// Mitsubishi GX Works2 project: 4way-intersection   PLC: Q03UDV

PROGRAM MAIN
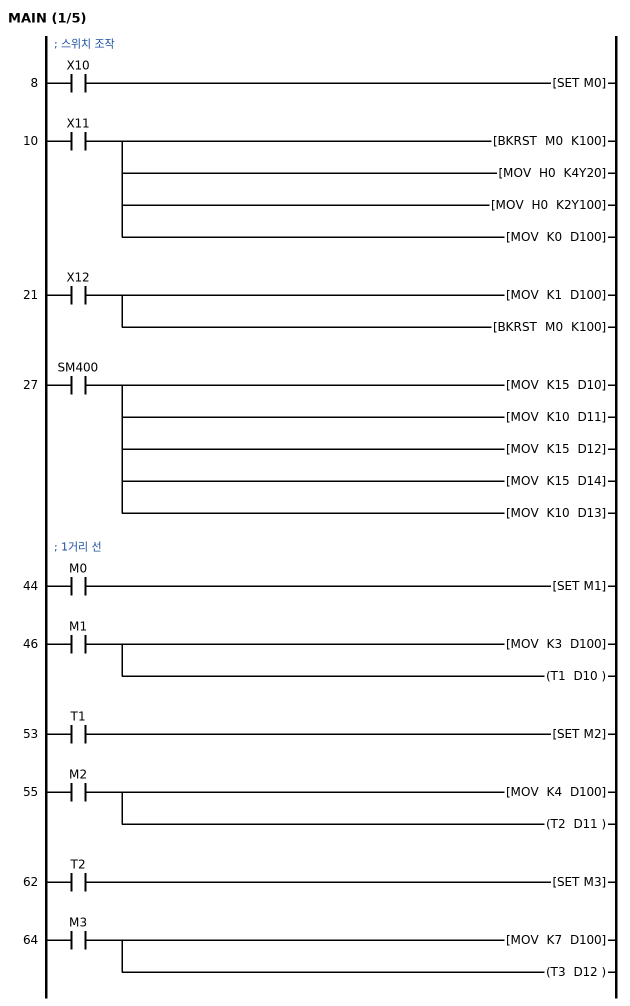
; 스위치 조작
8     LD      X10
      SET     M0
10    LD      X11
      BKRST   M0 K100
      MOV     H0 K4Y20
      MOV     H0 K2Y100
      MOV     K0 D100
21    LD      X12
      MOV     K1 D100
      BKRST   M0 K100
27    LD      SM400
      MOV     K15 D10
      MOV     K10 D11
      MOV     K15 D12
      MOV     K15 D14
      MOV     K10 D13
; 1거리 선
44    LD      M0
      SET     M1
46    LD      M1
      MOV     K3 D100
      OUT     T1 D10
53    LD      T1
      SET     M2
55    LD      M2
      MOV     K4 D100
      OUT     T2 D11
62    LD      T2
      SET     M3
64    LD      M3
      MOV     K7 D100
      OUT     T3 D12
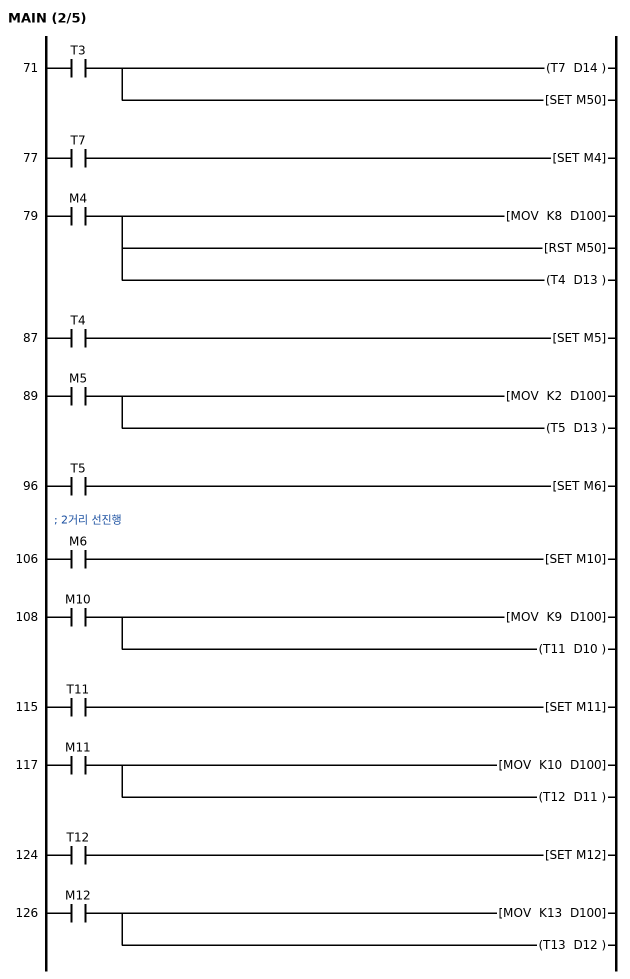
71    LD      T3
      OUT     T7 D14
      SET     M50
77    LD      T7
      SET     M4
79    LD      M4
      MOV     K8 D100
      RST     M50
      OUT     T4 D13
87    LD      T4
      SET     M5
89    LD      M5
      MOV     K2 D100
      OUT     T5 D13
96    LD      T5
      SET     M6
; 2거리 선진행
106   LD      M6
      SET     M10
108   LD      M10
      MOV     K9 D100
      OUT     T11 D10
115   LD      T11
      SET     M11
117   LD      M11
      MOV     K10 D100
      OUT     T12 D11
124   LD      T12
      SET     M12
126   LD      M12
      MOV     K13 D100
      OUT     T13 D12
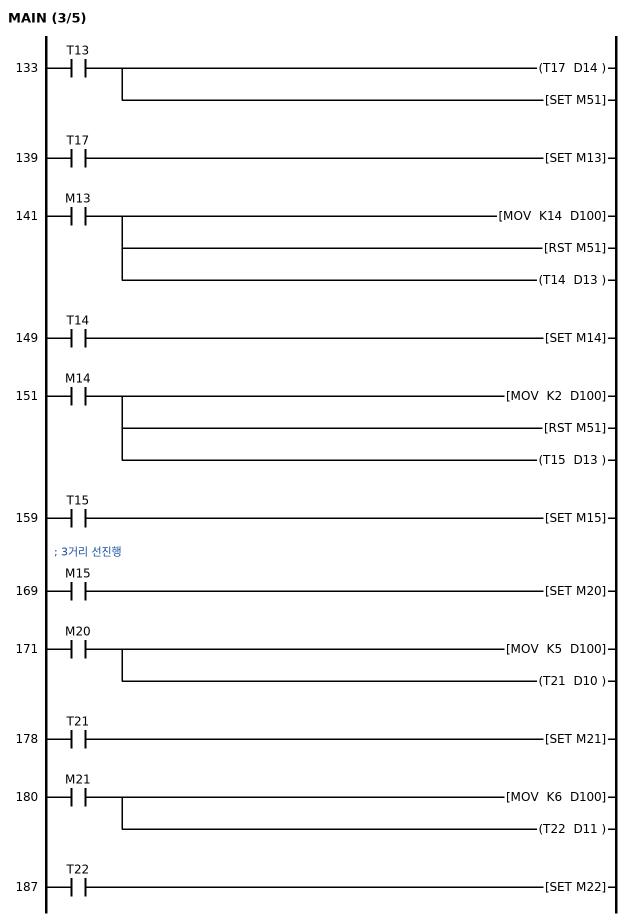
133   LD      T13
      OUT     T17 D14
      SET     M51
139   LD      T17
      SET     M13
141   LD      M13
      MOV     K14 D100
      RST     M51
      OUT     T14 D13
149   LD      T14
      SET     M14
151   LD      M14
      MOV     K2 D100
      RST     M51
      OUT     T15 D13
159   LD      T15
      SET     M15
; 3거리 선진행
169   LD      M15
      SET     M20
171   LD      M20
      MOV     K5 D100
      OUT     T21 D10
178   LD      T21
      SET     M21
180   LD      M21
      MOV     K6 D100
      OUT     T22 D11
187   LD      T22
      SET     M22
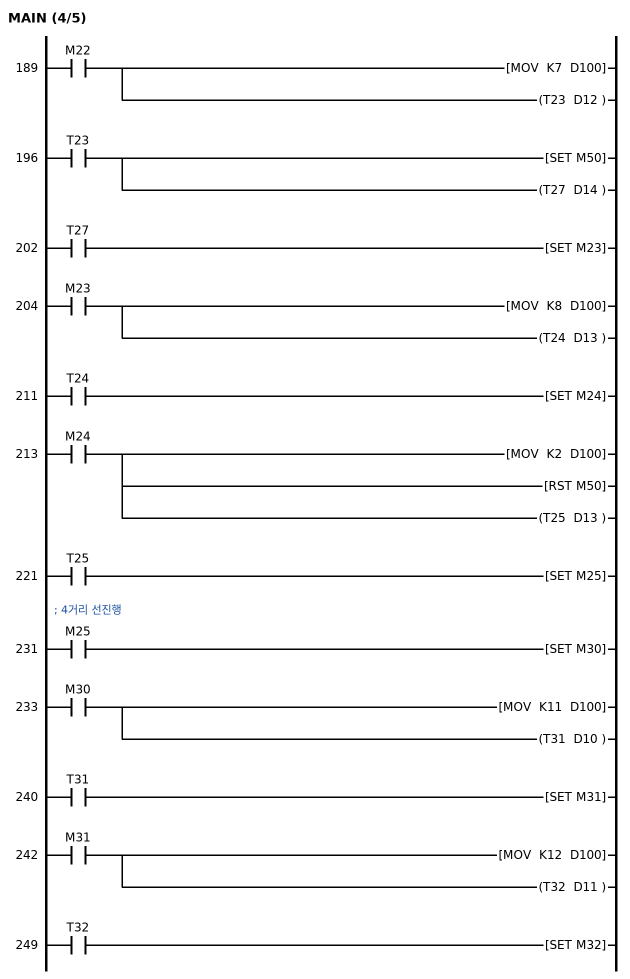
189   LD      M22
      MOV     K7 D100
      OUT     T23 D12
196   LD      T23
      SET     M50
      OUT     T27 D14
202   LD      T27
      SET     M23
204   LD      M23
      MOV     K8 D100
      OUT     T24 D13
211   LD      T24
      SET     M24
213   LD      M24
      MOV     K2 D100
      RST     M50
      OUT     T25 D13
221   LD      T25
      SET     M25
; 4거리 선진행
231   LD      M25
      SET     M30
233   LD      M30
      MOV     K11 D100
      OUT     T31 D10
240   LD      T31
      SET     M31
242   LD      M31
      MOV     K12 D100
      OUT     T32 D11
249   LD      T32
      SET     M32
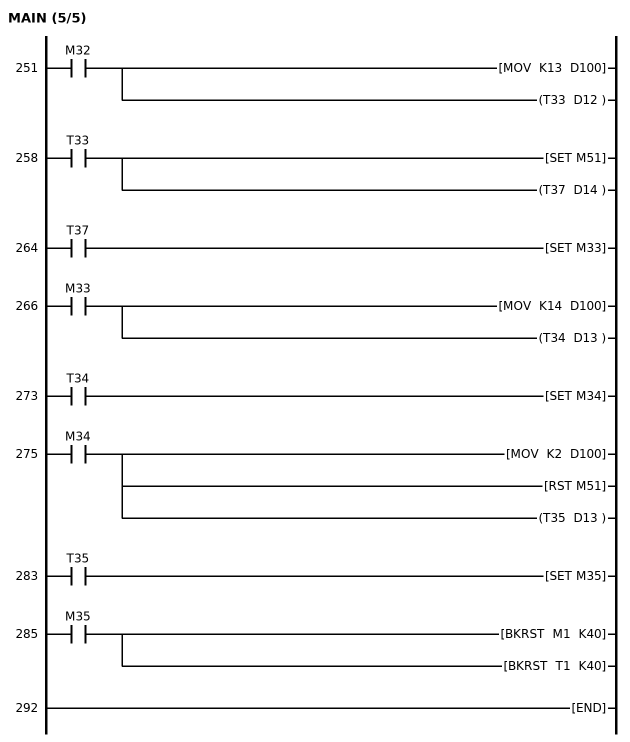
251   LD      M32
      MOV     K13 D100
      OUT     T33 D12
258   LD      T33
      SET     M51
      OUT     T37 D14
264   LD      T37
      SET     M33
266   LD      M33
      MOV     K14 D100
      OUT     T34 D13
273   LD      T34
      SET     M34
275   LD      M34
      MOV     K2 D100
      RST     M51
      OUT     T35 D13
283   LD      T35
      SET     M35
285   LD      M35
      BKRST   M1 K40
      BKRST   T1 K40
292   END
END_PROGRAM

PROGRAM HMI
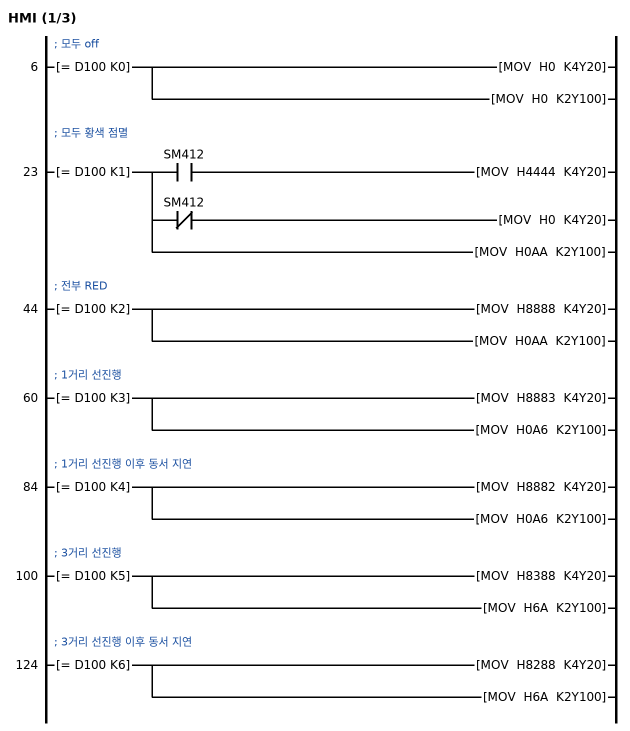
; 모두 off
6     LD=     D100 K0
      MOV     H0 K4Y20
      MOV     H0 K2Y100
; 모두 황색 점멸
23    LD=     D100 K1
      MPS
      AND     SM412
      MOV     H4444 K4Y20
      MRD
      ANI     SM412
      MOV     H0 K4Y20
      MPP
      MOV     H0AA K2Y100
; 전부 RED
44    LD=     D100 K2
      MOV     H8888 K4Y20
      MOV     H0AA K2Y100
; 1거리 선진행
60    LD=     D100 K3
      MOV     H8883 K4Y20
      MOV     H0A6 K2Y100
; 1거리 선진행 이후 동서 지연
84    LD=     D100 K4
      MOV     H8882 K4Y20
      MOV     H0A6 K2Y100
; 3거리 선진행
100   LD=     D100 K5
      MOV     H8388 K4Y20
      MOV     H6A K2Y100
; 3거리 선진행 이후 동서 지연
124   LD=     D100 K6
      MOV     H8288 K4Y20
      MOV     H6A K2Y100
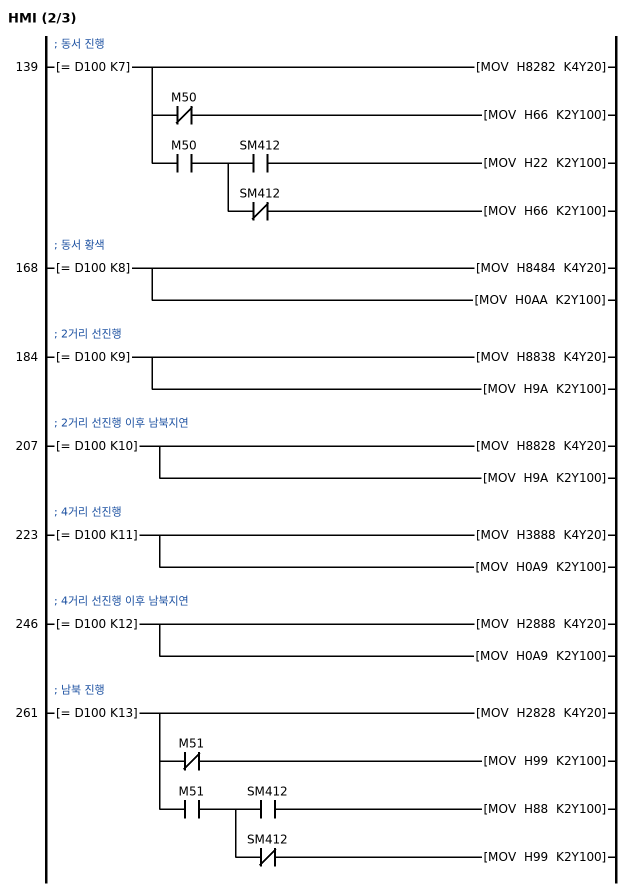
; 동서 진행
139   LD=     D100 K7
      MOV     H8282 K4Y20
      MPS
      ANI     M50
      MOV     H66 K2Y100
      MPP
      AND     M50
      MPS
      AND     SM412
      MOV     H22 K2Y100
      MPP
      ANI     SM412
      MOV     H66 K2Y100
; 동서 황색
168   LD=     D100 K8
      MOV     H8484 K4Y20
      MOV     H0AA K2Y100
; 2거리 선진행
184   LD=     D100 K9
      MOV     H8838 K4Y20
      MOV     H9A K2Y100
; 2거리 선진행 이후 남북지연
207   LD=     D100 K10
      MOV     H8828 K4Y20
      MOV     H9A K2Y100
; 4거리 선진행
223   LD=     D100 K11
      MOV     H3888 K4Y20
      MOV     H0A9 K2Y100
; 4거리 선진행 이후 남북지연
246   LD=     D100 K12
      MOV     H2888 K4Y20
      MOV     H0A9 K2Y100
; 남북 진행
261   LD=     D100 K13
      MOV     H2828 K4Y20
      MPS
      ANI     M51
      MOV     H99 K2Y100
      MPP
      AND     M51
      MPS
      AND     SM412
      MOV     H88 K2Y100
      MPP
      ANI     SM412
      MOV     H99 K2Y100
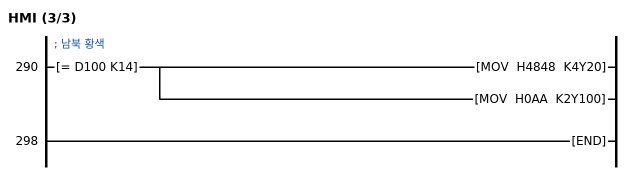
; 남북 황색
290   LD=     D100 K14
      MOV     H4848 K4Y20
      MOV     H0AA K2Y100
298   END
END_PROGRAM
